(* CoDeSys 2.3 export: MonitorDint.EXP *)

(* POU basic/MonitorDint, ST *)
FUNCTION MonitorDint : BOOL
VAR_INPUT
    Value: DINT;
    Channel: UINT;
END_VAR
VAR_IN_OUT
    Data: DINT;
END_VAR
VAR
END_VAR
IF Value <> Data THEN
    IF Channel < 256 THEN
        EvtCh8Tick32Int32(UINT_TO_BYTE(Channel), GlobalTick, Value, GlobalLogBufferHandle);
    ELSE
        EvtCh16Tick32Int32(Channel, GlobalTick, Value, GlobalLogBufferHandle);
    END_IF
    Data := Value;
END_IF
END_FUNCTION
